// SIMATIC STEP 7 (V5.x) project Линия сборки банки №1
// CPU: CPU 312
// station: Hardware
// station: SIMATIC 300(1)
// station: P_ADR_BUS
// station: P_ADR_BUS
// station: Configuration
// program: S7 Program(1)

SYMBOL_TABLE
"Банка №8"	FC 1	FC 1
"Банка №12"	FC 2	FC 2
"Сообщ. Банка №8"	FC 3	FC 3
"Сообщ. Банка №12"	FC 4	FC 4
"S1.1-S1.3"	I 0.0	BOOL	// Делитель. Защитный кожух.
"S1.4"	I 0.1	BOOL	// Делитель. Штурвал.
"S1.8-S1.9"	I 0.2	BOOL	// Делитель. Контроль брака на инструменте.
"S10-S12"	I 0.3	BOOL	// Делитель. Контроль замятия банок на выходе.
"S2.1-S2.3"	I 0.4	BOOL	// Отбортовка №1. Защитный кожух.
"S2.4"	I 0.5	BOOL	// Отбортовка №1. Штурвал.
"S3.1-S3.3"	I 0.6	BOOL	// Закатка №1. Защитный кожух.
"S3.4"	I 0.7	BOOL	// Закатка №1. Штурвал.
"S4.1"	I 1.0	BOOL	// Переключатель Б.№8--Б.№12
"S4.2"	I 1.1	BOOL	// Делитель. Вкл.
"S4.2a"	I 1.2	BOOL	// Делитель. Вкл. на закатке.
"S4.3-S4.3a"	I 1.3	BOOL	// Делитель. Откл.
"S4.4"	I 1.4	BOOL	// Отбортовка №1. Вкл.
"S4.4a"	I 1.5	BOOL	// Отбортовка №1. Вкл. на закатке.
"S4.5-S4.5a"	I 1.6	BOOL	// Отбортовка №1. Откл.
"S4.6"	I 1.7	BOOL	// Закатка №1. Вкл.
"S4.7"	I 2.0	BOOL	// Закатка №1. Откл.
"B1.5"	I 2.1	BOOL	// Давление воздуха.
"8B1"	I 2.2	BOOL	// Накопитель перед делителем. Минимум банки.
"8B2"	I 2.3	BOOL	// Счетчик +
"8B3"	I 2.4	BOOL	// Датчик такта.
"8B4"	I 2.5	BOOL	// Счетчик -. Левый выход.
"8B5"	I 2.6	BOOL	// Счетчик -. Правый выход.
"8B6"	I 2.7	BOOL	// Накопитель перед отбортовкой №1. Максимум банки.
"8B7"	I 3.0	BOOL	// Накопитель перед отбортовкой №1. Минимум банки.
"8B8"	I 3.1	BOOL	// Накопитель перед закаткой №1. Максимум банки.
"8B9"	I 3.2	BOOL	// Накопитель перед закаткой №1. Минимум банки.
"8B10"	I 3.3	BOOL	// Закатка №1. Подача крышки.
"S4.11"	I 3.4	BOOL	// Общий СТОП. Делитель,Отбортовка №1, Закатка №1.
"S4.8"	I 3.5	BOOL	// Делитель. Медленная прокрутка.
"S4.9"	I 3.6	BOOL	// Отбортовка №1. Медленная прокрутка.
"S4.10"	I 3.7	BOOL	// Закатка №1. Медленная прокрутка.
"8B11"	I 4.0	BOOL	// Накопитель перед отбортовкой №2. Минимум банки.
"8B12"	I 4.1	BOOL	// Накопитель перед закаткой №2. Максимум банки.
"8B13"	I 4.2	BOOL	// Накопитель перед закаткой №2. Минимум банки.
"8B14"	I 4.3	BOOL	// Закатка №2. Подача крышки.
"S5.1-S5.3"	I 4.4	BOOL	// Отбортовка №2. Защитный кожух.
"S5.4"	I 4.5	BOOL	// Отбортовка №2. Штурвал.
"S6.1-S6.3"	I 4.6	BOOL	// Закатка №2. Защитный кожух.
"S6.4"	I 4.7	BOOL	// Закатка №2. Штурвал.
"S7.1"	I 5.0	BOOL	// Отбортовка №2. Вкл.
"S7.1a"	I 5.1	BOOL	// Отбортовка №2. Вкл. на закатке №2.
"S7.2-S7.2a"	I 5.2	BOOL	// Отбортовка №2. Откл.
"S7.3"	I 5.3	BOOL	// Закатка №2. Вкл.
"S7.4"	I 5.4	BOOL	// Закатка №2. Откл.
"S7.5"	I 5.5	BOOL	// Общий СТОП. Отбортовка №2, Закатка №2.
"S7.6"	I 5.6	BOOL	// Отбортовка №2. Медленная прокрутка.
"S7.7"	I 5.7	BOOL	// Закатка №2. Медленная прокрутка.
"Y1.1"	Q 8.0	BOOL	// Эл.магнит подачи корпусов. Делитель.
"Y2.1"	Q 8.1	BOOL	// Эл.магнит подачи корпусов. Отбортовка №1.
"M1"	Q 8.2	BOOL	// Делитель.
"M3"	Q 8.3	BOOL	// Отбортовка №1.
"Y3.1"	Q 8.4	BOOL	// Эл.магнит подачи корпусов. Закатка №1.
"Y3.2"	Q 8.5	BOOL	// Эл.магнит подачи крышки.Закатка №1
"M1 JOG"	Q 8.6	BOOL	// Делитель.
"M3 JOG"	Q 8.7	BOOL	// Отбортовка №1.
"K9.7(M8)"	Q 12.0	BOOL	// Подъемник отбортовки №2.
"K9.8(M10)"	Q 12.1	BOOL	// Подъемник закатки №2.
"К9.9(М6)"	Q 12.2	BOOL	// Подъемник закатки №1.
"K9.5(M2)"	Q 12.4	BOOL	// Подъемник делителя.
"K9.6(M4)"	Q 12.5	BOOL	// Подъемник отбортовки №1.
"Y4.1"	Q 16.0	BOOL	// Эл.магнит подачи корпусов. Отбортовка №2.
"Y5.1"	Q 16.1	BOOL	// Эл.магнит подачи корпусов. Закатка №2.
"M7"	Q 16.2	BOOL	// Отбортовка №2.
"M7 JOG"	Q 16.3	BOOL	// Отбортовка №2.
"Y5.2"	Q 16.4	BOOL	// Эл.магнит подачи крышки.Закатка №2.
"M9"	Q 16.6	BOOL	// Закатка №2.
"M9 JOG"	Q 16.7	BOOL	// Закатка №2.
"M5"	Q 20.0	BOOL	// Закатка №1.
"M5 JOG"	Q 20.1	BOOL	// Закатка №1.
END_SYMBOL_TABLE

FUNCTION "Банка №8" : VOID	// FC 1
TITLE = Банка №8
VERSION : 0.1
BEGIN
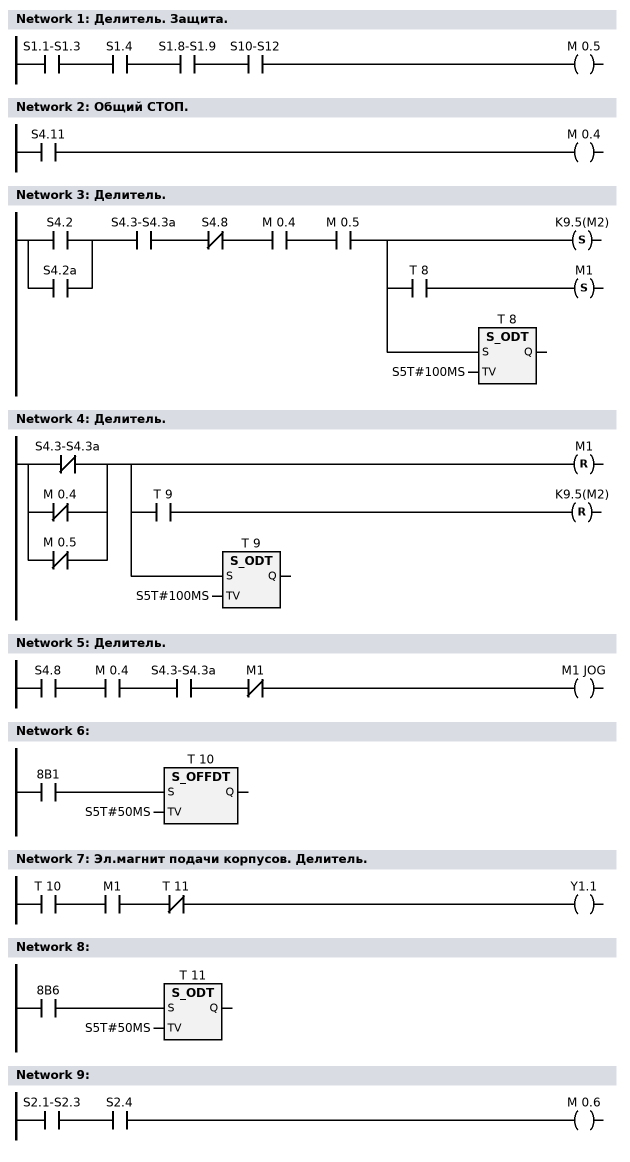
NETWORK
TITLE = Делитель. Защита.
      A     "S1.1-S1.3";
      A     "S1.4";
      A     "S1.8-S1.9";
      A     "S10-S12";
      =     M 0.5;
NETWORK
TITLE = Общий СТОП.
//На делитель, отбортовку №1, закатку №1.
      A     "S4.11";
      =     M 0.4;
NETWORK
TITLE = Делитель.
      A(;
      O     "S4.2";
      O     "S4.2a";
      );
      A     "S4.3-S4.3a";
      AN    "S4.8";
      A     M 0.4;
      A     M 0.5;
      =     L 0.0;
      A     L 0.0;
      BLD   102;
      S     "K9.5(M2)";
      A     L 0.0;
      A     T 8;
      S     "M1";
      A     L 0.0;
      L     S5T#100MS;
      SD    T 8;
      NOP   0;
      NOP   0;
      NOP   0;
      NOP   0;
NETWORK
TITLE = Делитель.
      ON    "S4.3-S4.3a";
      ON    M 0.4;
      ON    M 0.5;
      =     L 0.0;
      A     L 0.0;
      BLD   102;
      R     "M1";
      A     L 0.0;
      A     T 9;
      R     "K9.5(M2)";
      A     L 0.0;
      L     S5T#100MS;
      SD    T 9;
      NOP   0;
      NOP   0;
      NOP   0;
      NOP   0;
NETWORK
TITLE = Делитель.
//Медленная прокрутка.
      A     "S4.8";
      A     M 0.4;
      A     "S4.3-S4.3a";
      AN    "M1";
      =     "M1 JOG";
NETWORK
TITLE =
      A     "8B1";
      L     S5T#50MS;
      SF    T 10;
      NOP   0;
      NOP   0;
      NOP   0;
      NOP   0;
NETWORK
TITLE = Эл.магнит подачи корпусов. Делитель.
      A     T 10;
      A     "M1";
      AN    T 11;
      =     "Y1.1";
NETWORK
TITLE =
      A     "8B6";
      L     S5T#50MS;
      SD    T 11;
      NOP   0;
      NOP   0;
      NOP   0;
      NOP   0;
NETWORK
TITLE =
      A     "S2.1-S2.3";
      A     "S2.4";
      =     M 0.6;
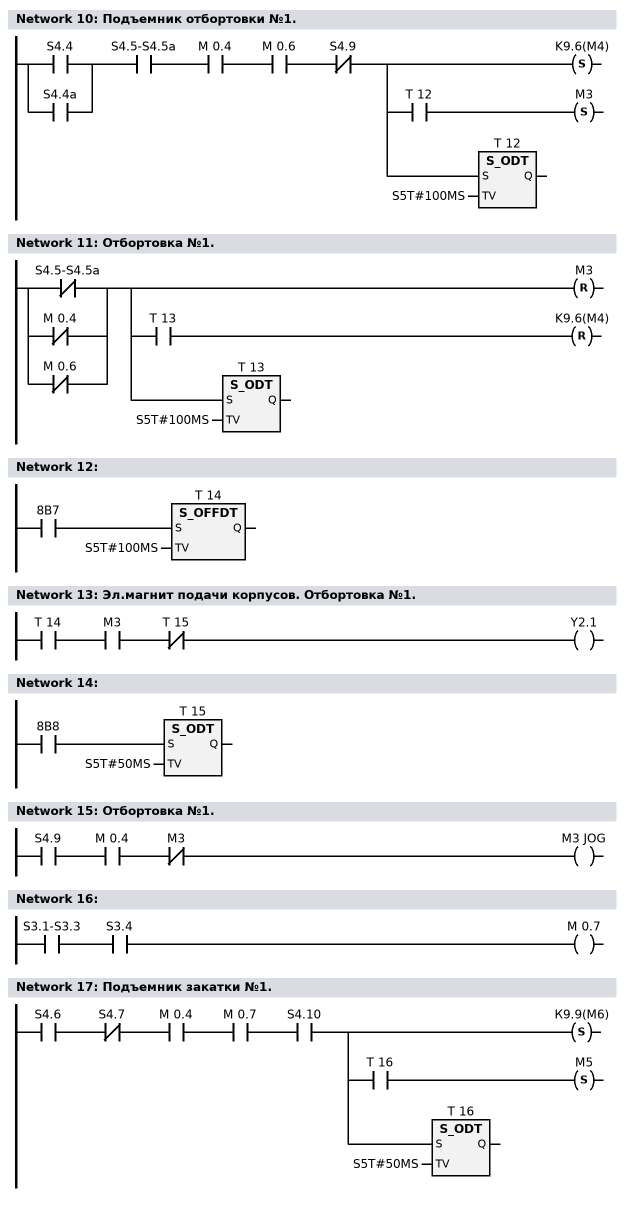
NETWORK
TITLE = Подъемник отбортовки №1.
      A(;
      O     "S4.4";
      O     "S4.4a";
      );
      A     "S4.5-S4.5a";
      A     M 0.4;
      A     M 0.6;
      AN    "S4.9";
      =     L 0.0;
      A     L 0.0;
      BLD   102;
      S     "K9.6(M4)";
      A     L 0.0;
      A     T 12;
      S     "M3";
      A     L 0.0;
      L     S5T#100MS;
      SD    T 12;
      NOP   0;
      NOP   0;
      NOP   0;
      NOP   0;
NETWORK
TITLE = Отбортовка №1.
      ON    "S4.5-S4.5a";
      ON    M 0.4;
      ON    M 0.6;
      =     L 0.0;
      A     L 0.0;
      BLD   102;
      R     "M3";
      A     L 0.0;
      A     T 13;
      R     "K9.6(M4)";
      A     L 0.0;
      L     S5T#100MS;
      SD    T 13;
      NOP   0;
      NOP   0;
      NOP   0;
      NOP   0;
NETWORK
TITLE =
      A     "8B7";
      L     S5T#100MS;
      SF    T 14;
      NOP   0;
      NOP   0;
      NOP   0;
      NOP   0;
NETWORK
TITLE = Эл.магнит подачи корпусов. Отбортовка №1.
      A     T 14;
      A     "M3";
      AN    T 15;
      =     "Y2.1";
NETWORK
TITLE =
      A     "8B8";
      L     S5T#50MS;
      SD    T 15;
      NOP   0;
      NOP   0;
      NOP   0;
      NOP   0;
NETWORK
TITLE = Отбортовка №1.
      A     "S4.9";
      A     M 0.4;
      AN    "M3";
      =     "M3 JOG";
NETWORK
TITLE =
      A     "S3.1-S3.3";
      A     "S3.4";
      =     M 0.7;
NETWORK
TITLE = Подъемник закатки №1.
      A     "S4.6";
      AN    "S4.7";
      A     M 0.4;
      A     M 0.7;
      A     "S4.10";
      =     L 0.0;
      A     L 0.0;
      BLD   102;
      S     "К9.9(М6)";
      A     L 0.0;
      A     T 16;
      S     "M5";
      A     L 0.0;
      L     S5T#50MS;
      SD    T 16;
      NOP   0;
      NOP   0;
      NOP   0;
      NOP   0;
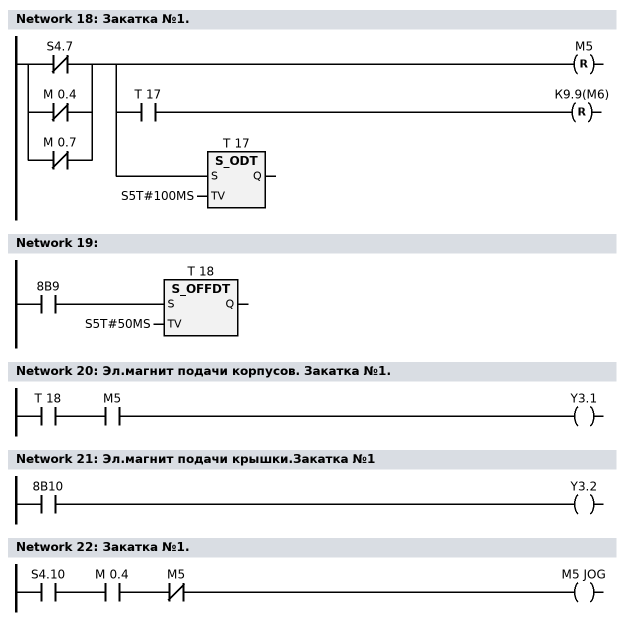
NETWORK
TITLE = Закатка №1.
      ON    "S4.7";
      ON    M 0.4;
      ON    M 0.7;
      =     L 0.0;
      A     L 0.0;
      BLD   102;
      R     "M5";
      A     L 0.0;
      A     T 17;
      R     "К9.9(М6)";
      A     L 0.0;
      L     S5T#100MS;
      SD    T 17;
      NOP   0;
      NOP   0;
      NOP   0;
      NOP   0;
NETWORK
TITLE =
      A     "8B9";
      L     S5T#50MS;
      SF    T 18;
      NOP   0;
      NOP   0;
      NOP   0;
      NOP   0;
NETWORK
TITLE = Эл.магнит подачи корпусов. Закатка №1.
      A     T 18;
      A     "M5";
      =     "Y3.1";
NETWORK
TITLE = Эл.магнит подачи крышки.Закатка №1
      A     "8B10";
      =     "Y3.2";
NETWORK
TITLE = Закатка №1.
      A     "S4.10";
      A     M 0.4;
      AN    "M5";
      =     "M5 JOG";
END_FUNCTION

FUNCTION "Банка №12" : VOID	// FC 2
TITLE = Банка №12
//Банка №12
VERSION : 0.1
BEGIN
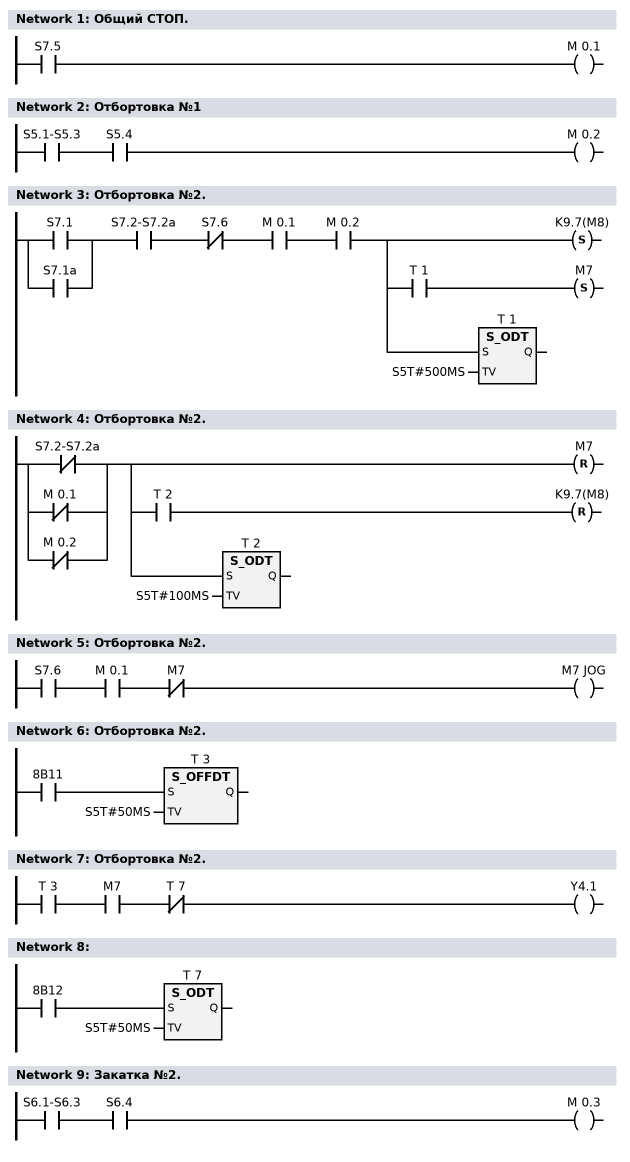
NETWORK
TITLE = Общий СТОП.
      A     "S7.5";
      =     M 0.1;
NETWORK
TITLE = Отбортовка №1
      A     "S5.1-S5.3";
      A     "S5.4";
      =     M 0.2;
NETWORK
TITLE = Oтбортовкa №2.
      A(;
      O     "S7.1";
      O     "S7.1a";
      );
      A     "S7.2-S7.2a";
      AN    "S7.6";
      A     M 0.1;
      A     M 0.2;
      =     L 0.0;
      A     L 0.0;
      BLD   102;
      S     "K9.7(M8)";
      A     L 0.0;
      A     T 1;
      S     "M7";
      A     L 0.0;
      L     S5T#500MS;
      SD    T 1;
      NOP   0;
      NOP   0;
      NOP   0;
      NOP   0;
NETWORK
TITLE = Отбортовка №2.
      ON    "S7.2-S7.2a";
      ON    M 0.1;
      ON    M 0.2;
      =     L 0.0;
      A     L 0.0;
      BLD   102;
      R     "M7";
      A     L 0.0;
      A     T 2;
      R     "K9.7(M8)";
      A     L 0.0;
      L     S5T#100MS;
      SD    T 2;
      NOP   0;
      NOP   0;
      NOP   0;
      NOP   0;
NETWORK
TITLE = Отбортовка №2.
//Медленная прокрутка.
      A     "S7.6";
      A     M 0.1;
      AN    "M7";
      =     "M7 JOG";
NETWORK
TITLE = Отбортовка №2.
      A     "8B11";
      L     S5T#50MS;
      SF    T 3;
      NOP   0;
      NOP   0;
      NOP   0;
      NOP   0;
NETWORK
TITLE = Отбортовка №2.
//Эл.магнит подачи корпусов.
      A     T 3;
      A     "M7";
      AN    T 7;
      =     "Y4.1";
NETWORK
TITLE =
      A     "8B12";
      L     S5T#50MS;
      SD    T 7;
      NOP   0;
      NOP   0;
      NOP   0;
      NOP   0;
NETWORK
TITLE = Закатка №2.
//Защита.
      A     "S6.1-S6.3";
      A     "S6.4";
      =     M 0.3;
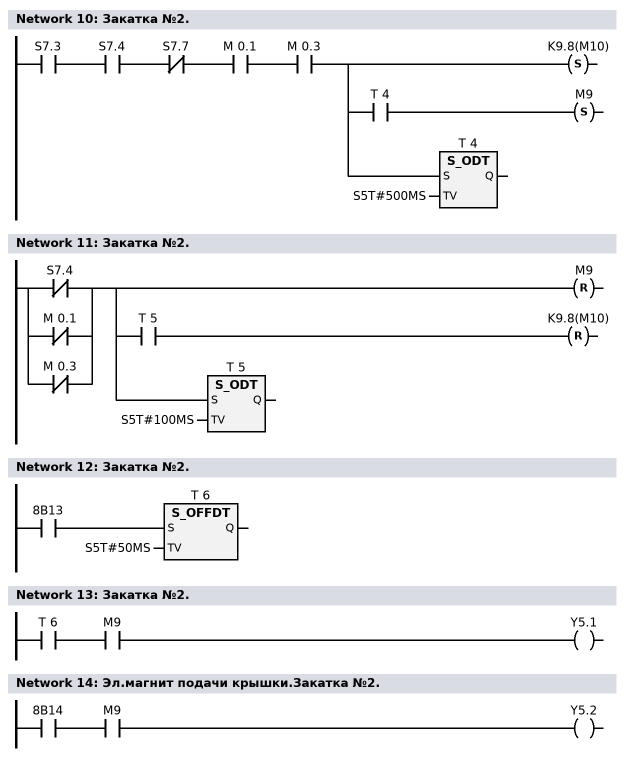
NETWORK
TITLE = Закатка №2.
      A     "S7.3";
      A     "S7.4";
      AN    "S7.7";
      A     M 0.1;
      A     M 0.3;
      =     L 0.0;
      A     L 0.0;
      BLD   102;
      S     "K9.8(M10)";
      A     L 0.0;
      A     T 4;
      S     "M9";
      A     L 0.0;
      L     S5T#500MS;
      SD    T 4;
      NOP   0;
      NOP   0;
      NOP   0;
      NOP   0;
NETWORK
TITLE = Закатка №2.
      ON    "S7.4";
      ON    M 0.1;
      ON    M 0.3;
      =     L 0.0;
      A     L 0.0;
      BLD   102;
      R     "M9";
      A     L 0.0;
      A     T 5;
      R     "K9.8(M10)";
      A     L 0.0;
      L     S5T#100MS;
      SD    T 5;
      NOP   0;
      NOP   0;
      NOP   0;
      NOP   0;
NETWORK
TITLE = Закатка №2.
      A     "8B13";
      L     S5T#50MS;
      SF    T 6;
      NOP   0;
      NOP   0;
      NOP   0;
      NOP   0;
NETWORK
TITLE = Закатка №2.
//Эл.магнит подачи корпусов. Закатка №2.
      A     T 6;
      A     "M9";
      =     "Y5.1";
NETWORK
TITLE = Эл.магнит подачи крышки.Закатка №2.
      A     "8B14";
      A     "M9";
      =     "Y5.2";
END_FUNCTION

FUNCTION "Сообщ. Банка №8" : VOID	// FC 3
//Сообщения: Банка №8.
VERSION : 0.1
BEGIN
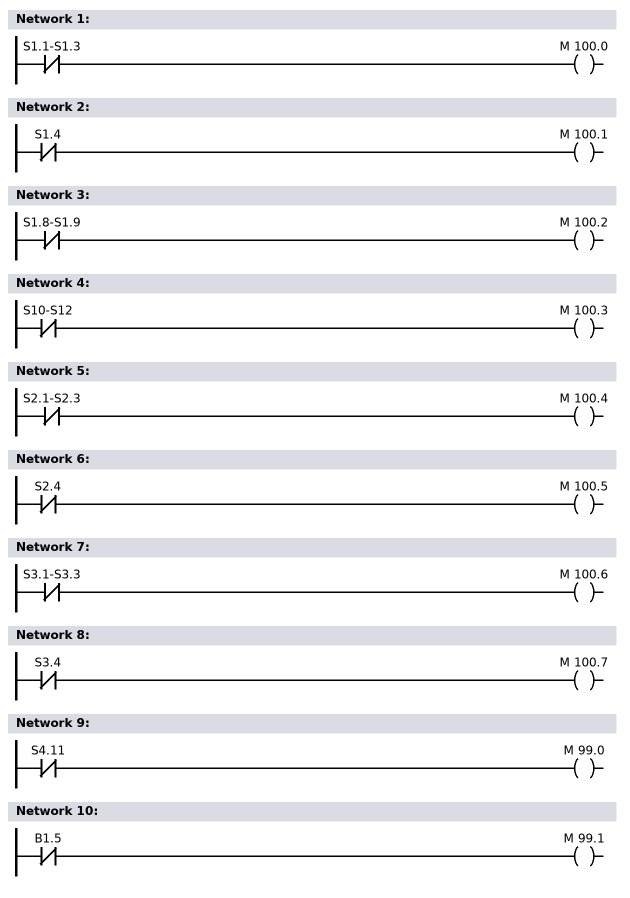
NETWORK
TITLE =
//Сообщение.Делитель.Защитный кожух открыт.
      AN    "S1.1-S1.3";
      =     M 100.0;
NETWORK
TITLE =
//Сообщение.Делитель.Штурвал в ручном режиме.
      AN    "S1.4";
      =     M 100.1;
NETWORK
TITLE =
//Сообщение.Делитель.Брак на инструменте.
      AN    "S1.8-S1.9";
      =     M 100.2;
NETWORK
TITLE =
//Сообщение.Делитель.Замята банка на выходе.
      AN    "S10-S12";
      =     M 100.3;
NETWORK
TITLE =
//Сообщение.Отбортовка №1.Защитный кожух открыт.
      AN    "S2.1-S2.3";
      =     M 100.4;
NETWORK
TITLE =
//Сообщение.Отбортовка №1.Штурвал в ручном режиме.
      AN    "S2.4";
      =     M 100.5;
NETWORK
TITLE =
//Сообщение.Закатка №1.Защитный кожух открыт.
      AN    "S3.1-S3.3";
      =     M 100.6;
NETWORK
TITLE =
//Сообщение.Закатка №1.Штурвал в ручном режиме.
      AN    "S3.4";
      =     M 100.7;
NETWORK
TITLE =
//Сообщение.Нажат общий СТОП на закатке.
      AN    "S4.11";
      =     M 99.0;
NETWORK
TITLE =
//Сообщение.Нет воздуха.
      AN    "B1.5";
      =     M 99.1;
END_FUNCTION

FUNCTION "Сообщ. Банка №12" : VOID	// FC 4
//Сообщения.Банка №12
VERSION : 0.1
BEGIN
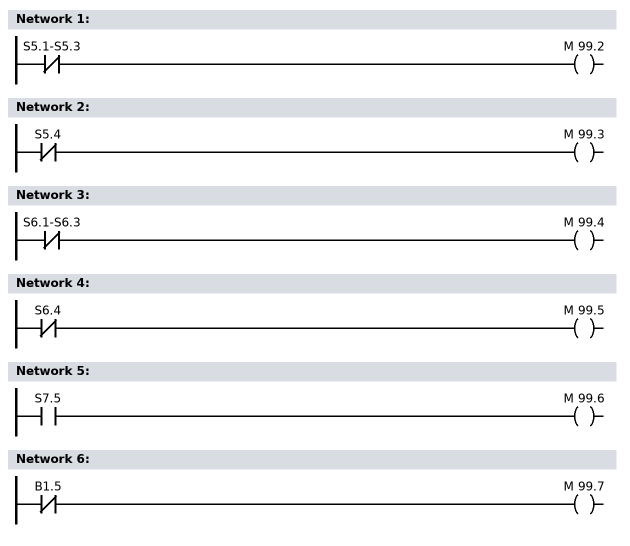
NETWORK
TITLE =
//Сообщение.Отбортовка №2.Защитный кожух открыт.
      AN    "S5.1-S5.3";
      =     M 99.2;
NETWORK
TITLE =
//Сообщение.Отбортовка №2.Штурвал в ручном режиме.
      AN    "S5.4";
      =     M 99.3;
NETWORK
TITLE =
//Сообщение.Закатка №2.Защитный кожух открыт.
      AN    "S6.1-S6.3";
      =     M 99.4;
NETWORK
TITLE =
//Сообщение.Закатка №2.Штурвал в ручном режиме.
      AN    "S6.4";
      =     M 99.5;
NETWORK
TITLE =
//Сообщение.Нет воздуха.
      A     "S7.5";
      =     M 99.6;
NETWORK
TITLE =
//Сообщение.
      AN    "B1.5";
      =     M 99.7;
END_FUNCTION

ORGANIZATION_BLOCK OB 1
TITLE = Организационный блок
VERSION : 0.1
VAR_TEMP
  OB1_EV_CLASS : BYTE ;	//Bits 0-3 = 1 (Coming event), Bits 4-7 = 1 (Event class 1)
  OB1_SCAN_1 : BYTE ;	//1 (Cold restart scan 1 of OB 1), 3 (Scan 2-n of OB 1)
  OB1_PRIORITY : BYTE ;	//Priority of OB Execution
  OB1_OB_NUMBR : BYTE ;	//1 (Organization block 1, OB1)
  OB1_RESERVED_1 : BYTE ;	//Reserved for system
  OB1_RESERVED_2 : BYTE ;	//Reserved for system
  OB1_PREV_CYCLE : INT ;	//Cycle time of previous OB1 scan (milliseconds)
  OB1_MIN_CYCLE : INT ;	//Minimum cycle time of OB1 (milliseconds)
  OB1_MAX_CYCLE : INT ;	//Maximum cycle time of OB1 (milliseconds)
  OB1_DATE_TIME : DATE_AND_TIME ;	//Date and time OB1 started
END_VAR
BEGIN
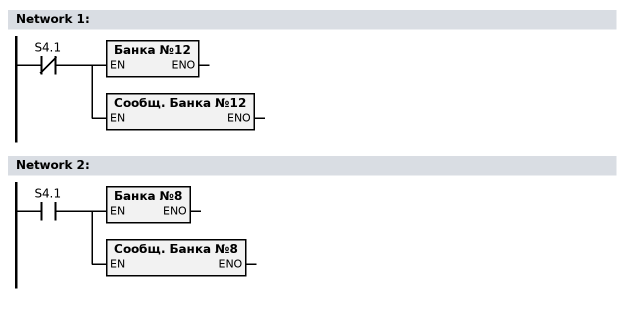
NETWORK
TITLE =
      AN    "S4.1";
      =     L 20.0;
      A     L 20.0;
      JNB   _001;
      CALL  "Банка №12";
_001: NOP   0;
      A     L 20.0;
      JNB   _004;
      CALL  "Сообщ. Банка №12";
_004: NOP   0;
NETWORK
TITLE =
      A     "S4.1";
      =     L 20.0;
      A     L 20.0;
      JNB   _005;
      CALL  "Банка №8";
_005: NOP   0;
      A     L 20.0;
      JNB   _006;
      CALL  "Сообщ. Банка №8";
_006: NOP   0;
END_ORGANIZATION_BLOCK
